// TIA Portal V15.1 export
// export: Created 2024-05-17T05:38:50.3568278Z, ExportSetting WithDefaults, DisplayName Totally Integrated Automation Portal, DisplayVersion V15.1 Update 5, DisplayName TIA Portal Openness, DisplayVersion V15.1 Update 5, DisplayName SINAMICS Startdrive Advanced, DisplayVersion V15.1, DisplayName G130, G150, S120, S150, SINAMICS MV, S210, DisplayVersion V15.1, DisplayName G110M, G120, G120C, G120D, G120P, DisplayVersion V15.1, DisplayName STEP 7 Professional, DisplayVersion V15.1 Update 5, DisplayName STEP 7 Safety, DisplayVersion V15.1, DisplayName WinCC Professional, DisplayVersion V15.1 Update 5, DisplayName SIMATIC Visualization Architect, DisplayVersion V15.1
FUNCTION_BLOCK "LGBLineConvBrake-MDXPN"   // FB6641, FBD
TITLE = LLineConvBrake-MDXPN
{ S7_Optimized_Access := 'TRUE' }
VERSION : 0.1
// stored: AutoNumber false, IsIECCheckEnabled false, IsRetainMemResEnabled false, MemoryReserve 100, SetENOAutomatically False, UDAEnableTagReadback false
   VAR_INPUT
      I_MotorProtection { ExternalAccessible := 'False'; ExternalVisible := 'False'; ExternalWritable := 'False'} : Bool;   // Motorprotection
      I_BrakeProtection { ExternalAccessible := 'False'; ExternalVisible := 'False'; ExternalWritable := 'False'} : Bool;   // Brake protection
      I_SafetySwitch { ExternalAccessible := 'False'; ExternalVisible := 'False'; ExternalWritable := 'False'} : Bool;   // Safety switch
      I_LocalPBSet { ExternalAccessible := 'False'; ExternalVisible := 'False'; ExternalWritable := 'False'} : Bool;   // Push button for manual movememt (on local panel)
      I_FncSelInHMIMain { ExternalAccessible := 'False'; ExternalVisible := 'False'; ExternalWritable := 'False'} : Bool;   // Function selected in HMI (From Main Drive)
      I_SafetyOk { ExternalAccessible := 'False'; ExternalVisible := 'False'; ExternalWritable := 'False'} : Bool;   // Safety Ok
      I_MotionStopOk { ExternalAccessible := 'False'; ExternalVisible := 'False'; ExternalWritable := 'False'} : Bool;   // Safety Ok / The motion stop is Ok
      I_SpeedMainDrive { ExternalAccessible := 'False'; ExternalVisible := 'False'; ExternalWritable := 'False'} : Int;   // Speed Value in mm/s
      I_EnabledriveCon { ExternalAccessible := 'False'; ExternalVisible := 'False'; ExternalWritable := 'False'} : Bool;   // Enable drive Condition
      I_ManSpeed { ExternalAccessible := 'False'; ExternalVisible := 'False'; ExternalWritable := 'False'} : Int;   // ManualSpeed Value in rpm
      I_SafetyStatusWord { ExternalAccessible := 'False'; ExternalVisible := 'False'; ExternalWritable := 'False'} : Word;   // Safety Status
      I_SafetyControlWord { ExternalAccessible := 'False'; ExternalVisible := 'False'; ExternalWritable := 'False'} : Word;   // Safety Control Word
   END_VAR
   VAR_OUTPUT
      O_Active { ExternalAccessible := 'False'; ExternalVisible := 'False'; ExternalWritable := 'False'} : Bool;   // Is Active
      O_ReadyForOperation { ExternalAccessible := 'False'; ExternalVisible := 'False'; ExternalWritable := 'False'} : Bool;   // Ready for operation
      O_EnableDrive { ExternalAccessible := 'False'; ExternalVisible := 'False'; ExternalWritable := 'False'} : Bool;   // Enable Drive
      O_AlarmABCondition { ExternalAccessible := 'False'; ExternalVisible := 'False'; ExternalWritable := 'False'} : Bool;   // Alarm AB condition
      O_AlarmA { ExternalAccessible := 'False'; ExternalVisible := 'False'; ExternalWritable := 'False'} : Bool;   // Alarm A
      O_AlarmB { ExternalAccessible := 'False'; ExternalVisible := 'False'; ExternalWritable := 'False'} : Bool;   // Alarm B
      O_AlarmC { ExternalAccessible := 'False'; ExternalVisible := 'False'; ExternalWritable := 'False'} : Bool;   // Alarm C
      O_AlarmD { ExternalAccessible := 'False'; ExternalVisible := 'False'; ExternalWritable := 'False'} : Bool;   // Alarm D
      H_AlarmWord { ExternalAccessible := 'False'; ExternalVisible := 'False'; ExternalWritable := 'False'} : DWord;   // Alarmword for WinCC
   END_VAR
   VAR_IN_OUT
      IO_Modes : "Modes";   // Modes
      H_HMI : "H_HMI";   // Animation
      "H_GBLineConvBrake-MDXPN" : "H_GBLineConvBrake-MDXPN";   // Animation
      C_Config : "LineConvBrake-MDXPNConfig";   // Config
   END_VAR
   VAR
      AA_MotorProtection { ExternalAccessible := 'False'; ExternalVisible := 'False'; ExternalWritable := 'False'} : Bool;   // Motor Protection Tripped
      AA_BrakeProtection { ExternalAccessible := 'False'; ExternalVisible := 'False'; ExternalWritable := 'False'} : Bool;   // Brake Protection Tripped
      AA_SafetySwitch { ExternalAccessible := 'False'; ExternalVisible := 'False'; ExternalWritable := 'False'} : Bool;   // Safety Switch Not Ok
      AB_Alarm { ExternalAccessible := 'False'; ExternalVisible := 'False'; ExternalWritable := 'False'} : Bool;   // Frequency Control Alarm
      AD_Warning { ExternalAccessible := 'False'; ExternalVisible := 'False'; ExternalWritable := 'False'} : Bool;   // Frequency Control Warning
      AD_MotionStop { ExternalAccessible := 'False'; ExternalVisible := 'False'; ExternalWritable := 'False'} : Bool;   // Motion Stop
      AC_ConfigRampAlm { ExternalAccessible := 'False'; ExternalVisible := 'False'; ExternalWritable := 'False'} : Bool;   // The config value for the ramp is not correct, must be zero or the config values for the calculation of the ramp must be ALL zero
      AC_ConfigRampCalcAlm { ExternalAccessible := 'False'; ExternalVisible := 'False'; ExternalWritable := 'False'} : Bool;   // The config values for the calculation of the ramp must be ALL different from zero
      SafetyOk { ExternalAccessible := 'False'; ExternalVisible := 'False'; ExternalWritable := 'False'} : Bool;   // Safety Ok
      MotorcmdSet { ExternalAccessible := 'False'; ExternalVisible := 'False'; ExternalWritable := 'False'} : Bool;   // Command High Speed to Motorloop set
      Speed { ExternalAccessible := 'False'; ExternalVisible := 'False'; ExternalWritable := 'False'} : Int;   // Speed Setting
      AlarmA { ExternalAccessible := 'False'; ExternalVisible := 'False'; ExternalWritable := 'False'} : Bool;   // Alarm A
      AlarmB { ExternalAccessible := 'False'; ExternalVisible := 'False'; ExternalWritable := 'False'} : Bool;   // Alarm B
      AlarmC { ExternalAccessible := 'False'; ExternalVisible := 'False'; ExternalWritable := 'False'} : Bool;   // Alarm C
      AlarmD { ExternalAccessible := 'False'; ExternalVisible := 'False'; ExternalWritable := 'False'} : Bool;   // Alarm D
      AlarmABCondition { ExternalAccessible := 'False'; ExternalVisible := 'False'; ExternalWritable := 'False'} : Bool;   // Alarm AB Condition
      ReadyForOperation { ExternalAccessible := 'False'; ExternalVisible := 'False'; ExternalWritable := 'False'} : Bool;   // Ready for operation
      MotorLoopActive { ExternalAccessible := 'False'; ExternalVisible := 'False'; ExternalWritable := 'False'} : Bool;   // Motor Loop Active
      MotorLoopAlarmCond { ExternalAccessible := 'False'; ExternalVisible := 'False'; ExternalWritable := 'False'} : Bool;   // Motor loop Alarm condition
      Edge { ExternalAccessible := 'False'; ExternalVisible := 'False'; ExternalWritable := 'False'} : Array[1..10] of Bool;   // Edge
      _LineConvBrake { ExternalAccessible := 'False'; ExternalVisible := 'False'; ExternalWritable := 'False'} : "LGBMotor2W2S-MDXPN-3PD";   // FB
   END_VAR
   VAR_TEMP
      H_HMIMotor : "H_HMI";   // Temp
   END_VAR
   VAR_TEMP   // added for the SCL form of the ladder/FBD networks
      _w1 : Bool;
   END_VAR
BEGIN

REGION Network 1: **** 1 - Inputs **** Safety Ok
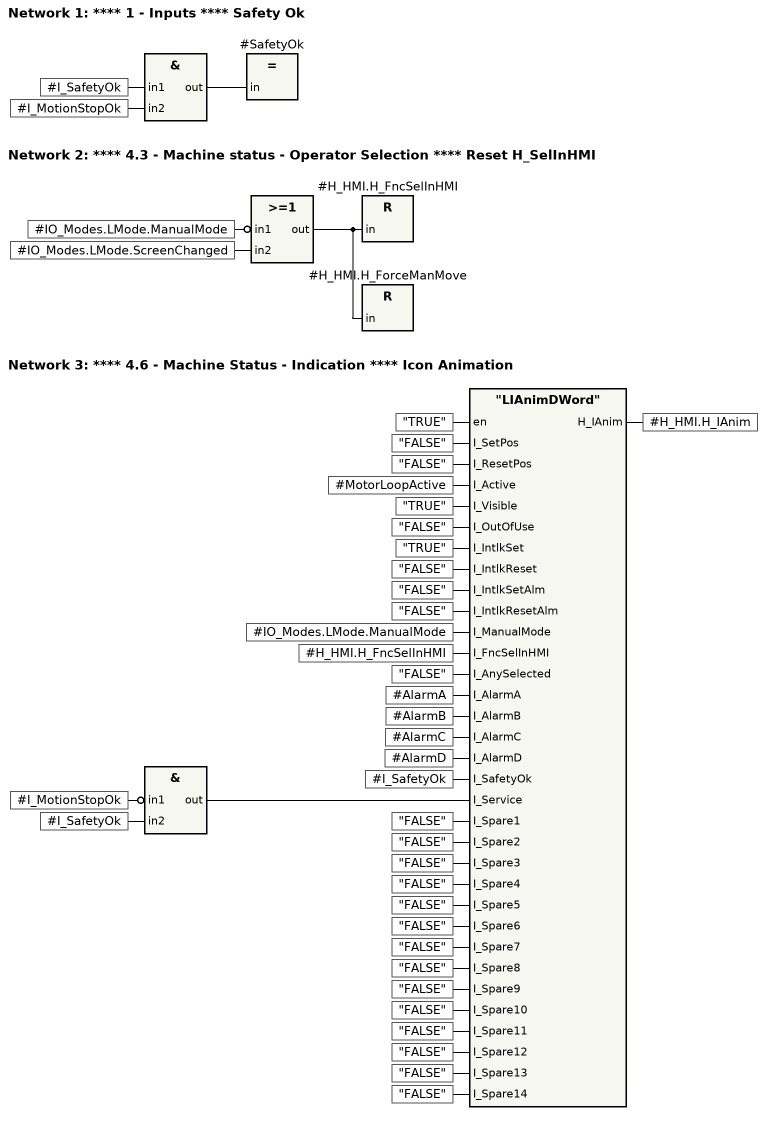
   #SafetyOk := #I_SafetyOk AND #I_MotionStopOk;
END_REGION

REGION Network 2: **** 4.3 - Machine status - Operator Selection **** Reset H_SelInHMI
   // Reset H_SelInHMI
   IF NOT #IO_Modes.LMode.ManualMode OR #IO_Modes.LMode.ScreenChanged THEN
       #H_HMI.H_FncSelInHMI := FALSE;
       #H_HMI.H_ForceManMove := FALSE;
   END_IF;
END_REGION

REGION Network 3: **** 4.6 - Machine Status - Indication **** Icon Animation
   // Icon Animation
   IF "TRUE" THEN
       "LIAnimDWord"(I_SetPos := "FALSE",
                     I_ResetPos := "FALSE",
                     I_Active := #MotorLoopActive,
                     I_Visible := "TRUE",
                     I_OutOfUse := "FALSE",
                     I_IntlkSet := "TRUE",
                     I_IntlkReset := "FALSE",
                     I_IntlkSetAlm := "FALSE",
                     I_IntlkResetAlm := "FALSE",
                     I_ManualMode := #IO_Modes.LMode.ManualMode,
                     I_FncSelInHMI := #H_HMI.H_FncSelInHMI,
                     I_AnySelected := "FALSE",
                     I_AlarmA := #AlarmA,
                     I_AlarmB := #AlarmB,
                     I_AlarmC := #AlarmC,
                     I_AlarmD := #AlarmD,
                     I_SafetyOk := #I_SafetyOk,
                     I_Service := NOT #I_MotionStopOk AND #I_SafetyOk,
                     I_Spare1 := "FALSE",
                     I_Spare2 := "FALSE",
                     I_Spare3 := "FALSE",
                     I_Spare4 := "FALSE",
                     I_Spare5 := "FALSE",
                     I_Spare6 := "FALSE",
                     I_Spare7 := "FALSE",
                     I_Spare8 := "FALSE",
                     I_Spare9 := "FALSE",
                     I_Spare10 := "FALSE",
                     I_Spare11 := "FALSE",
                     I_Spare12 := "FALSE",
                     I_Spare13 := "FALSE",
                     I_Spare14 := "FALSE",
                     H_IAnim => #H_HMI.H_IAnim);
   END_IF;
END_REGION

REGION Network 4: **** 4.6 - Machine Status - Indication **** Animation
   // Animation
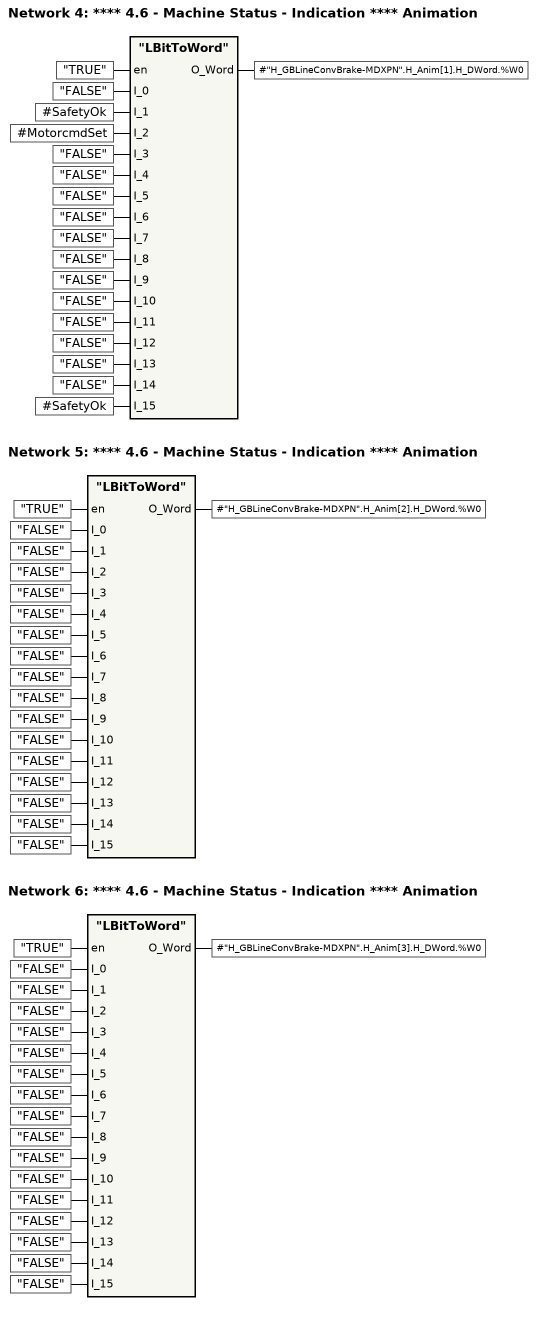
   IF "TRUE" THEN
       "LBitToWord"(I_0 := "FALSE",
                    I_1 := #SafetyOk,
                    I_2 := #MotorcmdSet,
                    I_3 := "FALSE",
                    I_4 := "FALSE",
                    I_5 := "FALSE",
                    I_6 := "FALSE",
                    I_7 := "FALSE",
                    I_8 := "FALSE",
                    I_9 := "FALSE",
                    I_10 := "FALSE",
                    I_11 := "FALSE",
                    I_12 := "FALSE",
                    I_13 := "FALSE",
                    I_14 := "FALSE",
                    I_15 := #SafetyOk,
                    O_Word => #"H_GBLineConvBrake-MDXPN".H_Anim[1].H_DWord.%W0);
   END_IF;
END_REGION

REGION Network 5: **** 4.6 - Machine Status - Indication **** Animation
   // Animation
   IF "TRUE" THEN
       "LBitToWord"(I_0 := "FALSE",
                    I_1 := "FALSE",
                    I_2 := "FALSE",
                    I_3 := "FALSE",
                    I_4 := "FALSE",
                    I_5 := "FALSE",
                    I_6 := "FALSE",
                    I_7 := "FALSE",
                    I_8 := "FALSE",
                    I_9 := "FALSE",
                    I_10 := "FALSE",
                    I_11 := "FALSE",
                    I_12 := "FALSE",
                    I_13 := "FALSE",
                    I_14 := "FALSE",
                    I_15 := "FALSE",
                    O_Word => #"H_GBLineConvBrake-MDXPN".H_Anim[2].H_DWord.%W0);
   END_IF;
END_REGION

REGION Network 6: **** 4.6 - Machine Status - Indication **** Animation
   // Animation
   IF "TRUE" THEN
       "LBitToWord"(I_0 := "FALSE",
                    I_1 := "FALSE",
                    I_2 := "FALSE",
                    I_3 := "FALSE",
                    I_4 := "FALSE",
                    I_5 := "FALSE",
                    I_6 := "FALSE",
                    I_7 := "FALSE",
                    I_8 := "FALSE",
                    I_9 := "FALSE",
                    I_10 := "FALSE",
                    I_11 := "FALSE",
                    I_12 := "FALSE",
                    I_13 := "FALSE",
                    I_14 := "FALSE",
                    I_15 := "FALSE",
                    O_Word => #"H_GBLineConvBrake-MDXPN".H_Anim[3].H_DWord.%W0);
   END_IF;
END_REGION

REGION Network 7: **** 4.6 - Machine Status - Indication **** Animation
   // Animation
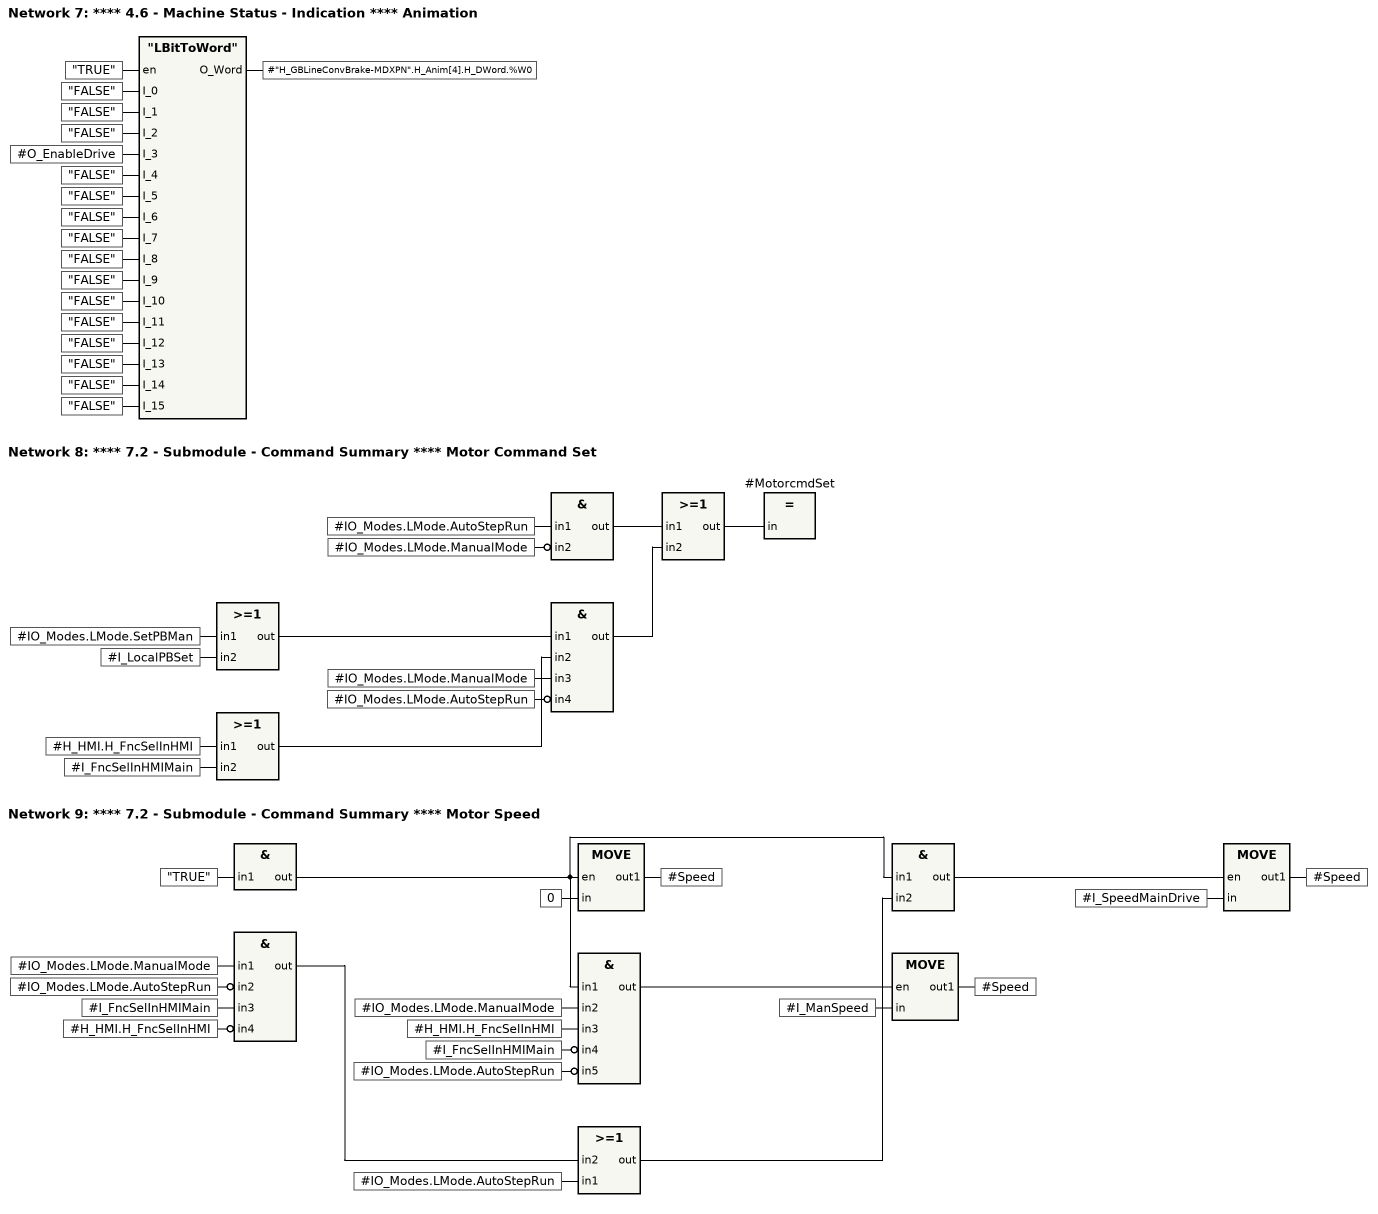
   IF "TRUE" THEN
       "LBitToWord"(I_0 := "FALSE",
                    I_1 := "FALSE",
                    I_2 := "FALSE",
                    I_3 := #O_EnableDrive,
                    I_4 := "FALSE",
                    I_5 := "FALSE",
                    I_6 := "FALSE",
                    I_7 := "FALSE",
                    I_8 := "FALSE",
                    I_9 := "FALSE",
                    I_10 := "FALSE",
                    I_11 := "FALSE",
                    I_12 := "FALSE",
                    I_13 := "FALSE",
                    I_14 := "FALSE",
                    I_15 := "FALSE",
                    O_Word => #"H_GBLineConvBrake-MDXPN".H_Anim[4].H_DWord.%W0);
   END_IF;
END_REGION

REGION Network 8: **** 7.2 - Submodule - Command Summary **** Motor Command Set
   // Motor Command
   #MotorcmdSet := (#IO_Modes.LMode.AutoStepRun AND NOT #IO_Modes.LMode.ManualMode) OR ((#IO_Modes.LMode.SetPBMan OR #I_LocalPBSet) AND (#H_HMI.H_FncSelInHMI OR #I_FncSelInHMIMain) AND #IO_Modes.LMode.ManualMode AND NOT #IO_Modes.LMode.AutoStepRun);
END_REGION

REGION Network 9: **** 7.2 - Submodule - Command Summary **** Motor Speed
   // Motor Speed
   IF "TRUE" THEN #Speed := 0; END_IF;
   IF "TRUE" AND #IO_Modes.LMode.ManualMode AND #H_HMI.H_FncSelInHMI AND NOT #I_FncSelInHMIMain AND NOT #IO_Modes.LMode.AutoStepRun THEN
       #Speed := #I_ManSpeed;
   END_IF;
   IF "TRUE" AND ((#IO_Modes.LMode.ManualMode AND NOT #IO_Modes.LMode.AutoStepRun AND #I_FncSelInHMIMain AND NOT #H_HMI.H_FncSelInHMI) OR #IO_Modes.LMode.AutoStepRun) THEN
       #Speed := #I_SpeedMainDrive;
   END_IF;
END_REGION

REGION Network 10: **** 7.3 - Submodule - Machine **** Motor loop MDXPN
   // Motor loop
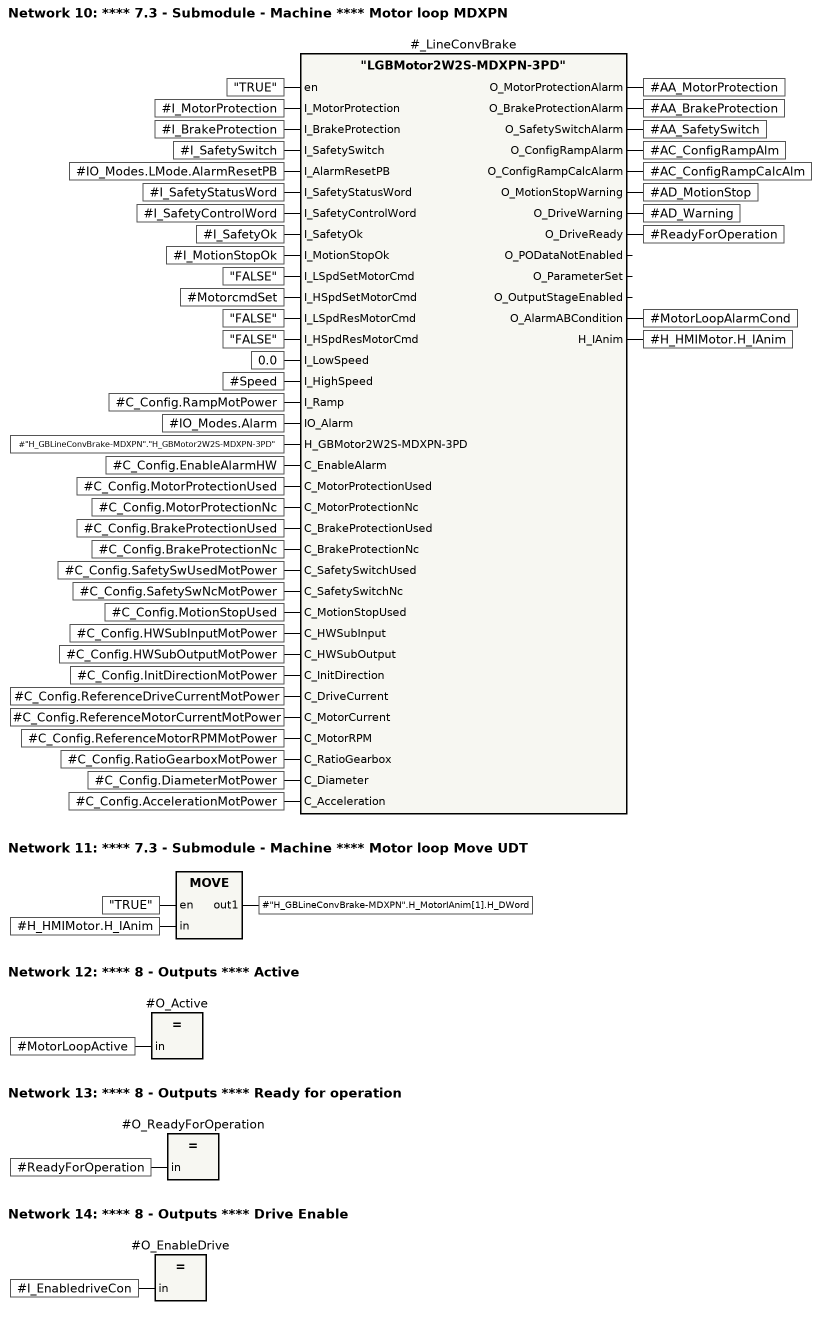
   IF "TRUE" THEN
       #_LineConvBrake(I_MotorProtection := #I_MotorProtection,   // "LGBMotor2W2S-MDXPN-3PD"
                       I_BrakeProtection := #I_BrakeProtection,
                       I_SafetySwitch := #I_SafetySwitch,
                       I_AlarmResetPB := #IO_Modes.LMode.AlarmResetPB,
                       I_SafetyStatusWord := #I_SafetyStatusWord,
                       I_SafetyControlWord := #I_SafetyControlWord,
                       I_SafetyOk := #I_SafetyOk,
                       I_MotionStopOk := #I_MotionStopOk,
                       I_LSpdSetMotorCmd := "FALSE",
                       I_HSpdSetMotorCmd := #MotorcmdSet,
                       I_LSpdResMotorCmd := "FALSE",
                       I_HSpdResMotorCmd := "FALSE",
                       I_LowSpeed := 0.0,
                       I_HighSpeed := #Speed,
                       I_Ramp := #C_Config.RampMotPower,
                       IO_Alarm := #IO_Modes.Alarm,
                       "H_GBMotor2W2S-MDXPN-3PD" := #"H_GBLineConvBrake-MDXPN"."H_GBMotor2W2S-MDXPN-3PD",
                       C_EnableAlarm := #C_Config.EnableAlarmHW,
                       C_MotorProtectionUsed := #C_Config.MotorProtectionUsed,
                       C_MotorProtectionNc := #C_Config.MotorProtectionNc,
                       C_BrakeProtectionUsed := #C_Config.BrakeProtectionUsed,
                       C_BrakeProtectionNc := #C_Config.BrakeProtectionNc,
                       C_SafetySwitchUsed := #C_Config.SafetySwUsedMotPower,
                       C_SafetySwitchNc := #C_Config.SafetySwNcMotPower,
                       C_MotionStopUsed := #C_Config.MotionStopUsed,
                       C_HWSubInput := #C_Config.HWSubInputMotPower,
                       C_HWSubOutput := #C_Config.HWSubOutputMotPower,
                       C_InitDirection := #C_Config.InitDirectionMotPower,
                       C_DriveCurrent := #C_Config.ReferenceDriveCurrentMotPower,
                       C_MotorCurrent := #C_Config.ReferenceMotorCurrentMotPower,
                       C_MotorRPM := #C_Config.ReferenceMotorRPMMotPower,
                       C_RatioGearbox := #C_Config.RatioGearboxMotPower,
                       C_Diameter := #C_Config.DiameterMotPower,
                       C_Acceleration := #C_Config.AccelerationMotPower,
                       O_MotorProtectionAlarm => #AA_MotorProtection,
                       O_BrakeProtectionAlarm => #AA_BrakeProtection,
                       O_SafetySwitchAlarm => #AA_SafetySwitch,
                       O_ConfigRampAlarm => #AC_ConfigRampAlm,
                       O_ConfigRampCalcAlarm => #AC_ConfigRampCalcAlm,
                       O_MotionStopWarning => #AD_MotionStop,
                       O_DriveWarning => #AD_Warning,
                       O_DriveReady => #ReadyForOperation,
                       O_AlarmABCondition => #MotorLoopAlarmCond,
                       H_IAnim => #H_HMIMotor.H_IAnim);
   END_IF;
END_REGION

REGION Network 11: **** 7.3 - Submodule - Machine **** Motor loop Move UDT
   IF "TRUE" THEN #"H_GBLineConvBrake-MDXPN".H_MotorIAnim[1].H_DWord := #H_HMIMotor.H_IAnim; END_IF;
END_REGION

REGION Network 12: **** 8 - Outputs **** Active
   // motor active
   #O_Active := #MotorLoopActive;
END_REGION

REGION Network 13: **** 8 - Outputs **** Ready for operation
   #O_ReadyForOperation := #ReadyForOperation;
END_REGION

REGION Network 14: **** 8 - Outputs **** Drive Enable
   #O_EnableDrive := #I_EnabledriveCon;
END_REGION

REGION Network 15: **** 8 - Outputs **** Alarm AB Condition
   // Alarm AB Condition
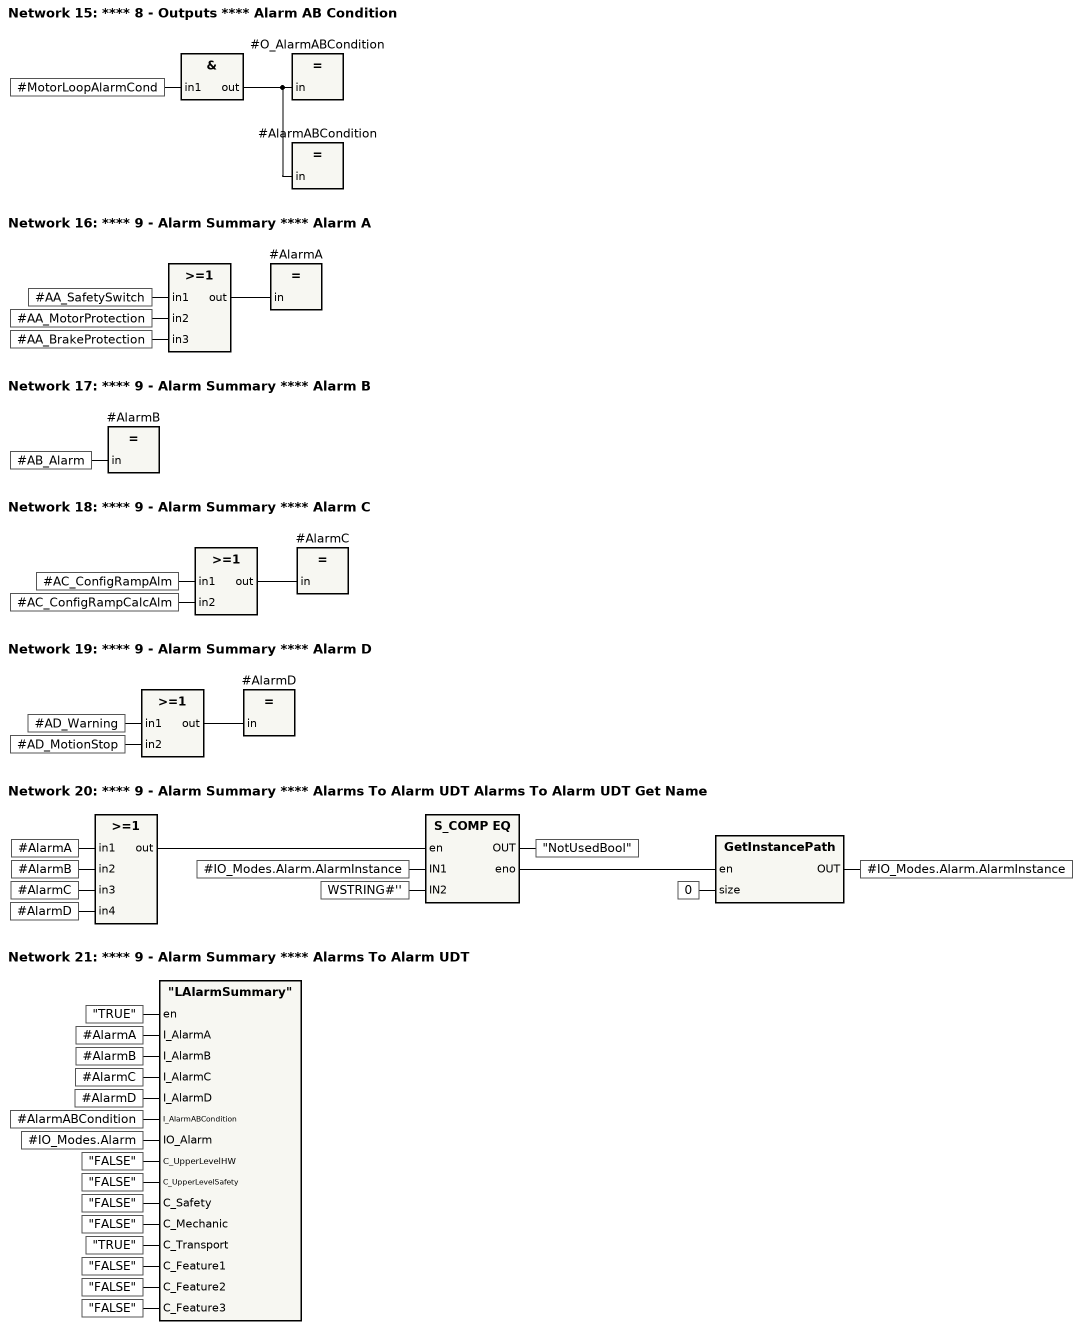
   #O_AlarmABCondition := #MotorLoopAlarmCond;
   #AlarmABCondition := #MotorLoopAlarmCond;
END_REGION

REGION Network 16: **** 9 - Alarm Summary **** Alarm A
   // Alarm A
   #AlarmA := #AA_SafetySwitch OR #AA_MotorProtection OR #AA_BrakeProtection;
END_REGION

REGION Network 17: **** 9 - Alarm Summary **** Alarm B
   // Alarm B
   #AlarmB := #AB_Alarm;
END_REGION

REGION Network 18: **** 9 - Alarm Summary **** Alarm C
   // Alarm C
   #AlarmC := #AC_ConfigRampAlm OR #AC_ConfigRampCalcAlm;
END_REGION

REGION Network 19: **** 9 - Alarm Summary **** Alarm D
   // Alarm D
   #AlarmD := #AD_Warning OR #AD_MotionStop;
END_REGION

REGION Network 20: **** 9 - Alarm Summary **** Alarms To Alarm UDT Alarms To Alarm UDT Get Name
   // Alarm D
   S_COMP(EN := #AlarmA OR #AlarmB OR #AlarmC OR #AlarmD,
          IN1 := #IO_Modes.Alarm.AlarmInstance,
          IN2 := WSTRING#'',
          OUT => "NotUsedBool",
          ENO => #_w1);
   IF #_w1 THEN GetInstancePath(size := 0, OUT => #IO_Modes.Alarm.AlarmInstance); END_IF;
END_REGION

REGION Network 21: **** 9 - Alarm Summary **** Alarms To Alarm UDT
   // Alarm D
   IF "TRUE" THEN
       "LAlarmSummary"(I_AlarmA := #AlarmA,
                       I_AlarmB := #AlarmB,
                       I_AlarmC := #AlarmC,
                       I_AlarmD := #AlarmD,
                       I_AlarmABCondition := #AlarmABCondition,
                       IO_Alarm := #IO_Modes.Alarm,
                       C_UpperLevelHW := "FALSE",
                       C_UpperLevelSafety := "FALSE",
                       C_Safety := "FALSE",
                       C_Mechanic := "FALSE",
                       C_Transport := "TRUE",
                       C_Feature1 := "FALSE",
                       C_Feature2 := "FALSE",
                       C_Feature3 := "FALSE");
   END_IF;
END_REGION

REGION Network 22: **** 9.1 - Alarm Output **** Alarm A
   // Alarm A
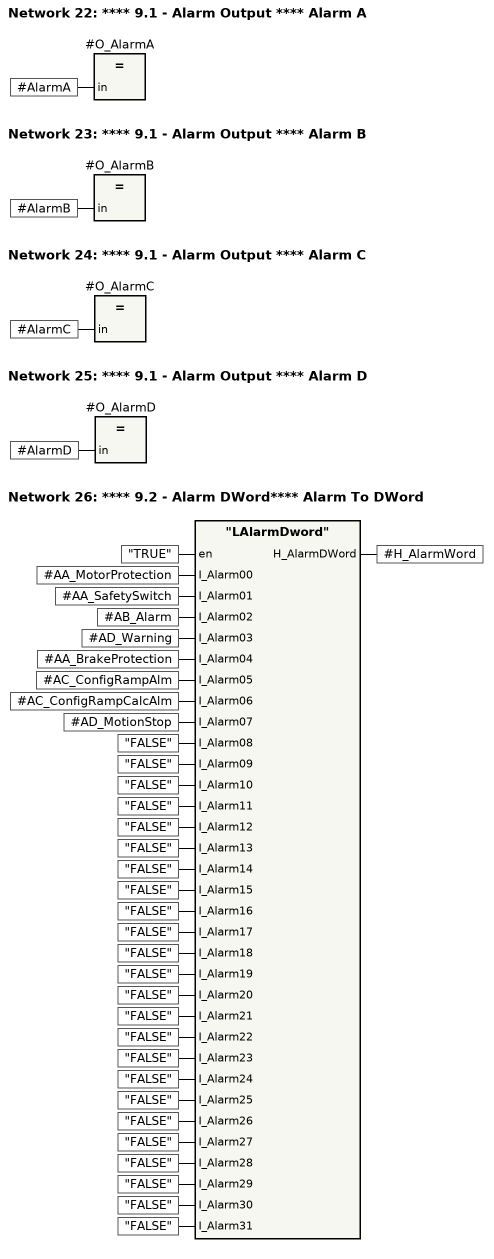
   #O_AlarmA := #AlarmA;
END_REGION

REGION Network 23: **** 9.1 - Alarm Output **** Alarm B
   // Alarm B
   #O_AlarmB := #AlarmB;
END_REGION

REGION Network 24: **** 9.1 - Alarm Output **** Alarm C
   // Alarm C
   #O_AlarmC := #AlarmC;
END_REGION

REGION Network 25: **** 9.1 - Alarm Output **** Alarm D
   // Alarm D
   #O_AlarmD := #AlarmD;
END_REGION

REGION Network 26: **** 9.2 - Alarm DWord**** Alarm To DWord
   // Alarm To Word
   IF "TRUE" THEN
       "LAlarmDword"(I_Alarm00 := #AA_MotorProtection,
                     I_Alarm01 := #AA_SafetySwitch,
                     I_Alarm02 := #AB_Alarm,
                     I_Alarm03 := #AD_Warning,
                     I_Alarm04 := #AA_BrakeProtection,
                     I_Alarm05 := #AC_ConfigRampAlm,
                     I_Alarm06 := #AC_ConfigRampCalcAlm,
                     I_Alarm07 := #AD_MotionStop,
                     I_Alarm08 := "FALSE",
                     I_Alarm09 := "FALSE",
                     I_Alarm10 := "FALSE",
                     I_Alarm11 := "FALSE",
                     I_Alarm12 := "FALSE",
                     I_Alarm13 := "FALSE",
                     I_Alarm14 := "FALSE",
                     I_Alarm15 := "FALSE",
                     I_Alarm16 := "FALSE",
                     I_Alarm17 := "FALSE",
                     I_Alarm18 := "FALSE",
                     I_Alarm19 := "FALSE",
                     I_Alarm20 := "FALSE",
                     I_Alarm21 := "FALSE",
                     I_Alarm22 := "FALSE",
                     I_Alarm23 := "FALSE",
                     I_Alarm24 := "FALSE",
                     I_Alarm25 := "FALSE",
                     I_Alarm26 := "FALSE",
                     I_Alarm27 := "FALSE",
                     I_Alarm28 := "FALSE",
                     I_Alarm29 := "FALSE",
                     I_Alarm30 := "FALSE",
                     I_Alarm31 := "FALSE",
                     H_AlarmDWord => #H_AlarmWord);
   END_IF;
END_REGION
END_FUNCTION_BLOCK
